PROGRAM MAIN
VAR
END_VAR

P_Inputs();
P_Filtering();
P_ControlBlock();
P_Output();
P_RunClock();

END_PROGRAM

(* stored: Version 1.1.0.1, ProductVersion 3.1.4024.13
   POU MAIN: Id {7af32e34-0e2b-468c-9d84-249dcd343744}, SpecialFunc None *)
